PROGRAM Get_Power
VAR
	voltage_effective : REAL;
	voltage_frequency : REAL;
	current_effective : REAL;
	current_frequency : REAL;
	power : REAL;
END_VAR

// Convert Data 

voltage_effective := INT_TO_REAL(gvl.gl_voltage_effective_raw)/65535*20; // Measured with an 
voltage_frequency := 1/(UINT_TO_REAL(gvl.gl_voltage_periode_raw)/1000); //convert ms to s and get Frequency from Period

current_effective := INT_TO_REAL(gvl.gl_current_effective_raw)/65535*20; // Measured with an 
current_frequency := 1/(UINT_TO_REAL(gvl.gl_current_periode_raw)/1000); //convert ms to s and get Frequency from Period

// Calculate Power 

power := voltage_effective * current_effective;

END_PROGRAM

(* stored: Version 1.1.0.1, ProductVersion 3.1.4024.12
   POU Get_Power: Id {1025fbe5-1567-453c-9968-b618e325114d}, SpecialFunc None *)
